// Core §7.7(c) — credential validation, injectable like every provider (§3.8).
// Returns the granted level; NONE = authentication failed. A provider may also
// implement I_AccessStore (a durable table), found by __QUERYINTERFACE.
INTERFACE I_AccessProvider EXTENDS __System.IQueryInterface

METHOD Authenticate : E_AccessLevel
VAR_INPUT
    User   : STRING(32);
    Secret : STRING(32);
END_VAR
END_METHOD

END_INTERFACE

(* stored: Version 1.1.0.1, ProductVersion 3.1.4024.12
   Itf I_AccessProvider: Id {02dbfd30-a6a4-4cc9-a8c8-fb07288e5b2e}
   Method Authenticate: Id {15290980-2c08-4c48-bfc3-81ef0d94a61f} *)
